{attribute 'GeneratedUsingTerminal: EL5151-0021-0018'}
{attribute addProperty BoxType "EL5151-0021-0018"}
{attribute addProperty Id "EtcSlaveTerminalBaseENC_StatusAT %I*ENC_Status_AC51C0C019ENC_Filtered_latchAT %I*ENC_Filtered_latch_2CF1EFF68ENC_ControlAT %Q*ENC_Control_EB66524120WcStateAT %I*WcState_9091E0EB2InfoDataAT %I*InfoData_32EB74EA10"}
{attribute addProperty CRC "242380241"}
{attribute addProperty Size "59"}
TYPE EL5151_0E726DD1 EXTENDS EtcSlaveTerminalBase :
STRUCT
	{attribute addProperty Name "ENC_Status"}
	ENC_Status : ENC_Status_AC51C0C0;
	{attribute addProperty Name "ENC_Filtered_latch"}
	ENC_Filtered_latch : ENC_Filtered_latch_2CF1EFF6;
	{attribute addProperty Name "ENC_Control"}
	ENC_Control : ENC_Control_EB665241;
	{attribute addProperty Name "WcState"}
	WcState : WcState_9091E0EB;
	{attribute addProperty Name "InfoData"}
	InfoData : InfoData_32EB74EA;
END_STRUCT
END_TYPE

(* stored: Version 1.2.0.0, ProductVersion 3.1.4024.9
   DUT EL5151_0E726DD1: Id {a3de8a67-8ea5-4101-ba7f-c4f2f1b34078} *)
